// TIA Portal V17 export
// export: Created 2024-09-02T12:50:31.622888Z, ExportSetting WithDefaults, DisplayName Totally Integrated Automation Portal, DisplayVersion V17, DisplayName TIA Portal Openness, DisplayVersion V17, DisplayName TIA Portal Version Control Interface, DisplayVersion V17, DisplayName STEP 7 Professional, DisplayVersion V17, DisplayName STEP 7 Safety, DisplayVersion V17, DisplayName WinCC Professional, DisplayVersion V17
TYPE "UFM_MovementParameters"
TITLE = UFM_MovementParameters
// Structure describing the parameter set for axis movements (for jog/move/wheel operations)
// stored: IsFailsafeCompliant false
   STRUCT
      Position : Real;   // Target position (irrelevant for wheel and jog)
      Speed : Real;   // Speed
      Overload : Real;   // Overload limit
      Signal : Real;   // Target signal for analog mode
      WheelRatio : Real;   // Wheel ratio
      Acceleration : Real;   // Acceleration
      OverloadSignalSource : Byte;   // Signal source for overload detection (sstNone .. sstLiveInput)
      OverloadComparisonOperator : Byte;   // Comparison operator to be used for overload detection (ocoGreaterOrEqual .. ocoGreaterOrEqualAbs)
      AnalogSignalSource : Byte;   // Signal source for analog mode (sstNone .. sstLiveInput)
      Mode : Byte;   // Movement mode (modePosition | modeAnalog)
      AnalogComparisonOperator : Byte;   // Comparison operator to be used for analog mode (ancoGreaterOrEqual | ancoLessOrEqual)
      AnalogTestDirection : Byte;   // Test direction for analog mode (tdDown | tdUp)
   END_STRUCT;
END_TYPE
